{attribute 'linkalways'} 
{attribute 'no_explicit_call' := 'This FB is a CLASS and must be accessed using methods or properties'}
{attribute 'enable_dynamic_creation'}
FUNCTION_BLOCK Node_F_VN_TransformIntoDisplayableImage EXTENDS VisionNode
VAR
    ipSrcImage : _ITcVnImage;
    ipDestImage : _ITcVnDisplayableImage;
    hrPrev : _HRESULT(S_OK);
	hresult : _HRESULT(S_OK);
END_VAR

METHOD PUBLIC  Clone : I_Node
VAR
	pNode : POINTER TO Node_F_VN_TransformIntoDisplayableImage;
END_VAR
pNode := __NEW(Node_F_VN_TransformIntoDisplayableImage);
Clone := pNode^;
END_METHOD

METHOD FB_init : BOOL
VAR_INPUT
	bInitRetains : BOOL; // if TRUE, the retain variables are initialized (warm start / cold start)
	bInCopyCode : BOOL;  // if TRUE, the instance afterwards gets moved into the copy code (online change)
END_VAR
AddInput('ipSrcImage', ipSrcImage);
AddInput('hrPrev', hrPrev);
AddOutput('ipDestImage', ipDestImage);
AddOutput('hresult',hresult);
END_METHOD

METHOD PROTECTED OnExecute
hresult.Value := F_VN_TransformIntoDisplayableImage(
    ipSrcImage := ipSrcImage.Value,
	ipDestImage := ipDestImage.Value,
	hrPrev:= hrPrev.Value);
END_METHOD

METHOD PUBLIC PreExecutionCheck
VAR_INPUT
	Check : I_PreExecutionChecks;
END_VAR
Check.IsTrue(ipSrcImage.IsValid, 'ipSrcImage must contain an image');
END_METHOD

END_FUNCTION_BLOCK

(* stored: Version 1.1.0.1, ProductVersion 3.1.4024.15
   POU Node_F_VN_TransformIntoDisplayableImage: Id {fdaaf4c1-57a0-0698-2205-93ff97b1852a}, SpecialFunc None
   Folder Constructor: Id {c3ffac90-f319-02c9-110f-9cd9b33586e3}
   Method Clone: Id {447c6bd3-1500-0ff9-3b45-8381f870915a}
   Method FB_init: Id {dfec66f4-d0ea-044c-22a5-9bfc94229ec4}
   Method OnExecute: Id {c64b7978-fa51-065d-2093-d0485b5ee08d}
   Method PreExecutionCheck: Id {f1b5fbc5-b2e7-0280-3896-457cd4f081c3} *)
